TYPE ST_EnclosureClimate_get :
STRUCT
	r_Humidity			: REAL;
	r_Temperature		: REAL;
	
	events				: ST_EnclosureClimate_events;
END_STRUCT
END_TYPE

(* stored: Version 1.1.0.1, ProductVersion 3.1.4024.12
   DUT ST_EnclosureClimate_get: Id {ce95f478-866a-47ba-b67e-bc5ac03966e0} *)
